// TIA Portal project "ISA_P10" (V16)

(* hardware
DEVICE "S7-1200 station_1"  S7-1200 Station
   slot 0: "Rack_0"  S7-1200 Rack  Rack  V1.0
   slot 1: "PLC_1"  CPU 1215C DC/DC/DC  6ES7 215-1AG40-0XB0  V4.4
DEVICE "Dispositivo GSD_1"  GSD.Device.PN
   slot 0: "FQ2"  FQ2-XXX  FQ2-XXX  1.9.0
      slot 0: "FQ2-XXX"  FQ2-XXX  1.9.0
      slot 1: "Output Data_1"  Output Data  1.9.0
         slot 0: "Output Data"  Output Data  1.9.0
      slot 1: "Interface"  Interface
         slot 1: "Port 1"  Port 1
   slot 0: "Rack"  Rack  V1.0
   slot 2: "Results Data - 32 items_1"  Results Data - 32 items  1.9.0
      slot 0: "Results Data - 32 items"  Results Data - 32 items  1.9.0
DEVICE "PC-System_1"  SIMATIC PC station
   slot 0: "Estación PC SIMATIC"  Rail  SIMATIC PC-Station  V1.0
      slot 125: "Stationmanager"  Station_Manager  V6.0.4
   slot 1: "HMI_RT_1"  WinCC RT Advanced  6AV2 104-0xxxx-xxxx  16.0.0.0
      slot 33792: "Interfaz del equipo"  Host interface
   slot 2: "IE general_1"  IE General  IE_CP  V8.2.0
*)

// ===== PLC "PLC_1"  CPU 1215C DC/DC/DC =====

VAR_GLOBAL   // PLC tag table "Tabla de variables estándar"
   "FQ2_Juicio" AT %ID84 : DWord;
   "FQ2_R" AT %ID88 : DWord;
   "FQ2_G" AT %ID92 : DWord;
   "FQ2_B" AT %ID96 : DWord;
   "FQ2_Trigger" AT %Q2.1 : Bool;
   "Pulsador_Trigger" AT %I0.0 : Bool;
END_VAR

DATA_BLOCK "Variables"   // DB1
{ S7_Optimized_Access := 'TRUE' }
VERSION : 0.1
   VAR
      rojo : Bool;
      green : Bool;
      blue : Bool;
      color : SInt;
   END_VAR
BEGIN
END_DATA_BLOCK

ORGANIZATION_BLOCK "Main"   // OB1, LAD, ProgramCycle
TITLE = "Main Program Sweep (Cycle)"
{ S7_Optimized_Access := 'TRUE' }
VERSION : 0.1
   VAR_INPUT
      Initial_Call : Bool;   // Initial call of this OB
      Remanence : Bool;   // =True, if remanent data are available
   END_VAR
BEGIN

REGION Network 1
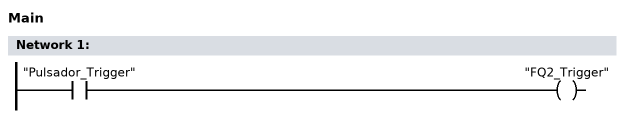
   RUNG wire#powerrail
      Contact( "Pulsador_Trigger" )
      Coil( "FQ2_Trigger" )
   END_RUNG
   // the same network as SCL:
   "FQ2_Trigger" := "Pulsador_Trigger";
END_REGION

REGION Network 2 (SCL)
   IF "FQ2_R" > 160000 AND "FQ2_G" < 70000 AND "FQ2_B" < 70000 THEN
       "Variables".color := 1;
   ELSIF "FQ2_R" < 80000 AND "FQ2_G" > 88000 AND "FQ2_B" < 70000 THEN
       "Variables".color := 2;
   ELSIF "FQ2_R" < 90000 AND "FQ2_G" < 100000 AND "FQ2_B" > 120000 THEN
       "Variables".color := 3;
   END_IF;
END_REGION
END_ORGANIZATION_BLOCK

(* ===== HMI "HMI_RT_1" =====
connection "HMI_Conexión_1": ETHERNET, S7_1200_OMS

HMI tags "Tabla de variables estándar"
   "Variables_color" : SInt = PLC Variables.color, 1 s

screen "Imagen_1" 800x600
   Circle "Círculo_1" at 180,53 size 427x427
      Appearance <- "Variables_color"
*)